{attribute addProperty BoxType "AT2041-0250-0020"}
{attribute addProperty Id "A_0102_AT2041_5250_0019_AT2041_5250AT2041_C5E5984862678.25"}
{attribute addProperty CRC "3003436130"}
{attribute addProperty SizeInBites "626"}
{attribute addProperty SizeInBytes "78.25"}
TYPE A_0042_AT2041_0250_0020_B304CC62 EXTENDS AT2041_BA5A9548 :
STRUCT
	{attribute addProperty Name "A_0102_AT2041_5250_0019_AT2041_5250"}
	A_0102_AT2041_5250_0019_AT2041_5250 : AT2041_C5E59848;
END_STRUCT
END_TYPE

(* stored: Version 1.2.0.0, ProductVersion 3.1.4024.9
   DUT A_0042_AT2041_0250_0020_B304CC62: Id {0c251815-29ae-44ca-b3df-2e918e8bee82} *)
